FUNCTION_BLOCK StopAerate (* Basic Function Block Type *)
  (* Standard: 61499-2 *)
  (* Version 0.0, 7/16/2026, Schneider Electric, Template *)
  PACKAGE SE.Nereda;
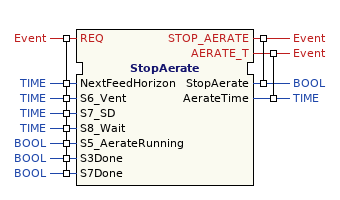
  EVENT_INPUT
    REQ WITH NextFeedHorizon, S6_Vent, S7_SD, S8_Wait, S5_AerateRunning, S3Done, S7Done; (* Normal Execution Request *)
  END_EVENT
  EVENT_OUTPUT
    STOP_AERATE WITH StopAerate; (* Execution Confirmation *)
    AERATE_T WITH AerateTime;
  END_EVENT
  VAR_INPUT
    NextFeedHorizon : TIME;
    S6_Vent : TIME;
    S7_SD : TIME;
    S8_Wait : TIME;
    S5_AerateRunning : BOOL;
    S3Done : BOOL;
    S7Done : BOOL;
  END_VAR
  VAR_OUTPUT
    StopAerate : BOOL;
    AerateTime : TIME;
  END_VAR
  VAR
    VentTime : REAL;
    SDTime : REAL;
    WaitTime : REAL;
    InNextFeedHorizon : REAL;
    SumState : REAL;
  END_VAR
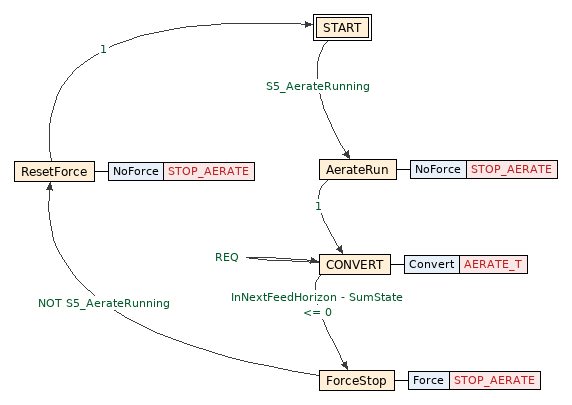
  EC_STATES
    START; (* Initial State *)
    AerateRun : NoForce -> STOP_AERATE;
    ForceStop : Force -> STOP_AERATE;
    ResetForce : NoForce -> STOP_AERATE;
    CONVERT : Convert -> AERATE_T;
  END_STATES
  EC_TRANSITIONS
    START TO AerateRun := S5_AerateRunning;
    CONVERT TO ForceStop := InNextFeedHorizon - SumState <= 0;
    ForceStop TO ResetForce := NOT S5_AerateRunning;
    ResetForce TO START := 1;
    AerateRun TO CONVERT := 1;
    CONVERT TO CONVERT := REQ;
  END_TRANSITIONS
  ALGORITHM NoForce IN ST:
;
StopAerate := FALSE;
  END_ALGORITHM
  ALGORITHM Force IN ST:
;
StopAerate := TRUE;
  END_ALGORITHM
  ALGORITHM Convert IN ST:
;
VentTime := TIME_TO_REAL(S6_Vent / 1000);
SDTime := TIME_TO_REAL(S7_SD / 1000);
WaitTime := TIME_TO_REAL(S8_Wait / 1000);
InNextFeedHorizon := TIME_TO_REAL(NextFeedHorizon / 1000);

IF S3Done THEN
	SumState := VentTime + WaitTime;
ELSE
	SumState := VentTime + SDTime + WaitTime;
END_IF;

AerateTime := REAL_TO_TIME((InNextFeedHorizon - SumState) * 1000);
  END_ALGORITHM
END_FUNCTION_BLOCK
